// TwinCAT 3 PLC project Factory_Method_Pattern
// ProgramVersion: 3.1.4024.0
// libraries:
//   Tc2_Standard, * (Beckhoff Automation GmbH)
//   Tc2_System, * (Beckhoff Automation GmbH)
//   Tc3_Module, * (Beckhoff Automation GmbH)
// project tree:
//   Classes/ BasicObject.TcPOU, ITF_Cyclic.TcIO, ITF_Mover.TcIO, ITF_Station.TcIO, ITF_Track.TcIO, Mover.TcPOU, Station.TcPOU, Track.TcPOU
//   FactoryBase/ Factory.TcPOU, ITF_Factory.TcIO
//   Factorys/ MoverFactory.TcPOU, StationFactory.TcPOU, TrackFactory.TcPOU
//   / PlcTask.TcTTO
//   POUs/ MAIN.TcPOU
// (motion and I/O tree: see PLC project simple_factory_pattern)
// real-time tasks:
//   TASK PlcTask: cycle T#10ms, priority 20, ADS port 350
//   TASK PlcTask1: cycle T#10ms, priority 21, ADS port 351
//   TASK PlcTask2: cycle T#10ms, priority 22, ADS port 352
//   TASK PlcTask3: cycle T#10ms, priority 23, ADS port 353
//   TASK PlcTask4: cycle T#10ms, priority 24, ADS port 354
//   TASK PlcTask5: cycle T#10ms, priority 25, ADS port 355
//   TASK PlcTask6: cycle T#10ms, priority 26, ADS port 356
//   TASK PlcTask7: cycle T#10ms, priority 27, ADS port 357
//   TASK PlcTask8: cycle T#10ms, priority 28, ADS port 358
//   TASK PlcTask9: cycle T#10ms, priority 29, ADS port 359
//   TASK PlcTask10: cycle T#10ms, priority 30, ADS port 360
//   TASK PlcTask11: cycle T#10ms, priority 31, ADS port 361

CONFIGURATION Factory_Method_Pattern
    RESOURCE PLC ON TwinCAT3
        TASK PlcTask(INTERVAL := T#10ms, PRIORITY := 21);
        PROGRAM MAIN WITH PlcTask : MAIN;
    END_RESOURCE
END_CONFIGURATION

// ---- Classes/ITF_Cyclic.TcIO
INTERFACE ITF_Cyclic EXTENDS __SYSTEM.IQueryInterface

METHOD Cycle : BOOL
VAR_INPUT
END_VAR
END_METHOD

END_INTERFACE

// ---- Classes/ITF_Mover.TcIO
INTERFACE ITF_Mover

METHOD MaxVelo : BOOL
VAR_INPUT
	MaxVelocity : LREAL;
END_VAR
END_METHOD

END_INTERFACE

// ---- Classes/ITF_Station.TcIO
INTERFACE ITF_Station

METHOD Position : BOOL;
VAR_INPUT
	StationPosition : LREAL;
END_VAR
END_METHOD

END_INTERFACE

// ---- Classes/ITF_Track.TcIO
INTERFACE ITF_Track

METHOD Length : BOOL
VAR_INPUT
	TrackLength : LREAL;
END_VAR
END_METHOD

END_INTERFACE

// ---- FactoryBase/ITF_Factory.TcIO
INTERFACE ITF_Factory

METHOD Create : ITF_Cyclic
VAR_INPUT
END_VAR
END_METHOD

END_INTERFACE

// ---- POUs/MAIN.TcPOU
PROGRAM MAIN
VAR
	State: INT;
	XtsMoverFactory : MoverFactory;
	XtsStationFactory : StationFactory;
	XtsTrackFactory : TrackFactory;
	iFactory : ITF_Factory := XtsMoverFactory;
	XtsElements : ARRAY[0..8] OF ITF_Cyclic;
END_VAR

CASE State OF
	0:
		IF Initialise() THEN
			State := 1;
		END_IF
END_CASE

METHOD Initialise : BOOL
VAR_INPUT
END_VAR

VAR
	i: INT;
END_VAR
FOR i := 0 TO 2 DO
	XtsElements[i] := iFactory.Create();
END_FOR
iFactory := XtsStationFactory;
FOR i := 3 TO 5 DO
	XtsElements[i] := iFactory.Create();
END_FOR
iFactory := XtsTrackFactory;
FOR i := 6 TO 8 DO
	XtsElements[i] := iFactory.Create();
END_FOR
Initialise := TRUE;
END_METHOD

END_PROGRAM

// ---- Factorys/MoverFactory.TcPOU
FUNCTION_BLOCK MoverFactory EXTENDS Factory
VAR
	ptrMover : POINTER TO Mover;
	itfMover : ITF_Mover;
END_VAR

METHOD Create : ITF_Cyclic
VAR_INPUT
END_VAR
PtrMover := __NEW(Mover);
Create := ptrMover^;
IF __QUERYINTERFACE(Create,itfMover) THEN
	itfMover.MaxVelo(MaxVelocity := 4000.0);
END_IF
END_METHOD

END_FUNCTION_BLOCK

// ---- FactoryBase/Factory.TcPOU
FUNCTION_BLOCK Factory IMPLEMENTS ITF_Factory
VAR
	ObjPtr : POINTER TO BasicObject;
END_VAR

METHOD Create : ITF_Cyclic
VAR_INPUT
END_VAR
ObjPtr := __NEW(BasicObject);
Create := ObjPtr^;
END_METHOD

END_FUNCTION_BLOCK

// ---- Classes/BasicObject.TcPOU
{attribute 'enable_dynamic_creation'}
FUNCTION_BLOCK BasicObject IMPLEMENTS ITF_Cyclic
VAR_INPUT
END_VAR
VAR_OUTPUT
END_VAR
VAR
END_VAR

{warning 'add method implementation '}
METHOD Cycle : BOOL
END_METHOD

END_FUNCTION_BLOCK

// ---- Classes/Mover.TcPOU
{attribute 'enable_dynamic_creation'}
FUNCTION_BLOCK Mover IMPLEMENTS ITF_Cyclic, ITF_Mover
VAR
	myMaxVelo : LREAL;
END_VAR

{warning 'add method implementation '}
METHOD Cycle : BOOL
END_METHOD

METHOD MaxVelo : BOOL
VAR_INPUT
	MaxVelocity : LREAL;
END_VAR
END_METHOD

END_FUNCTION_BLOCK

// ---- Factorys/StationFactory.TcPOU
FUNCTION_BLOCK StationFactory EXTENDS Factory
VAR
	prtStation : POINTER TO Station;
	itfStation : ITF_Station;
END_VAR

METHOD Create : ITF_Cyclic
VAR_INPUT
END_VAR
prtStation := __NEW(Station);
Create := prtStation^;
IF __QUERYINTERFACE(Create,itfStation) THEN
	itfStation.Position(StationPosition := 1250.0);
END_IF
END_METHOD

END_FUNCTION_BLOCK

// ---- Classes/Station.TcPOU
{attribute 'enable_dynamic_creation'}
FUNCTION_BLOCK Station IMPLEMENTS ITF_Cyclic, ITF_Station
VAR
	MyTrackPosition : LREAL;
END_VAR

{warning 'add method implementation '}
METHOD Cycle : BOOL
END_METHOD

METHOD Position : BOOL
VAR_INPUT
	StationPosition	: LREAL;
END_VAR
MyTrackPosition := StationPosition;
END_METHOD

END_FUNCTION_BLOCK

// ---- Factorys/TrackFactory.TcPOU
FUNCTION_BLOCK TrackFactory EXTENDS Factory
VAR
	ptrTrack : POINTER TO Track;
	itfTrack : ITF_Track;
END_VAR

METHOD Create : ITF_Cyclic
VAR_INPUT
END_VAR
ptrTrack := __NEW(Track);
Create := ptrTrack^;
IF __QUERYINTERFACE(Create,itfTrack) THEN
	itfTrack.Length(TrackLength := 2500.0);
END_IF
END_METHOD

END_FUNCTION_BLOCK

// ---- Classes/Track.TcPOU
{attribute 'enable_dynamic_creation'}
FUNCTION_BLOCK Track IMPLEMENTS ITF_Cyclic, ITF_Track
VAR
	MyTrackLength : LREAL;
END_VAR

{warning 'add method implementation '}
METHOD Cycle : BOOL
END_METHOD

METHOD Length : bool
VAR_INPUT
	TrackLength : LREAL;
END_VAR
MyTrackLength := TrackLength;
END_METHOD

END_FUNCTION_BLOCK
